(* IEC 61131-3 sources: xpxp/llama3-8b, 17 files *)

(* ---- 15.st ---- *)
FUNCTION FC1002 :BOOL
VAR_INPUT
	E_A, SENSOR: BOOL;
	ZEITW: TIME;
END_VAR
VAR
	zeit := 0;
END_VAR
VAR_IN_OUT
	ZEIT: TON;
	P_HU, P_AL: BOOL;
END_VAR

IF E_A THEN
	IF SENSOR THEN
		zeit := TIMET#(ZEITW);
		LOOP zeit < 3000 DO
			P_HU := TRUE;
			TIMET#(ZEIT) +:= 100; // Simulate sensor update (100ms)
		REPEAT
		ELOOP
		P_AL := FALSE;
		zeit := TIMET#(ZEITW);
	END_IF
ELSIF zeit > 0 THEN
	P_AL := TRUE;
ELSE
	P_HU := FALSE;
	P_AL := FALSE;
ENDIF

(* ---- 18.st ---- *)
FUNCTION FC1003 : VOID
VAR_INPUT
    IN_R:REAL;
    IN_MAX, IN_MIN:REAL;
    OUT_MAX, OUT_MIN:REAL;
END_VAR
VAR_OUTPUT
    OUT_R:REAL;
    FEH:BOOL;
END_VAR
VAR_TEMP
    DIFF1, DIFF2:REAL;
END_VAR

OUT_R := (IN_R - IN_MIN) / (IN_MAX - IN_MIN) * (OUT_MAX - OUT_MIN) + OUT_MIN;

IF OUT_R < OUT_MIN THEN
    OUT_R := OUT_MIN;
ELSIF OUT_R > OUT_MAX THEN
    OUT_R := OUT_MAX;
END_IF;

FEH := TRUE;
END_FUNCTION;

(* ---- 19.st ---- *)
FUNCTION_BLOCK FB1005

VAR_INPUT
    START: BOOL;
    DICKE: REAL;
    V_MAX: REAL;
    V_MIN: REAL;
END_VAR

VAR_OUTPUT
    D_MAX: REAL;
    D_MIN: REAL;
    P1: BOOL;
END_VAR

VAR
    FO: BOOL;
    M_MAX: REAL;
    M_MIN: REAL;
    THICKNESS: REAL;
END_VAR

PROGRAM
    IF START THEN
        M_MAX := 0.0;
        M_MIN := 0.0;
    END_IF;

    IF DICKE > 0.0 THEN
        THICKNESS := ABS(DICKE - (V_MAX + V_MIN) / 2.0);
        IF THICKNESS > M_MAX THEN
            M_MAX := THICKNESS;
        END_IF;
        IF THICKNESS < M_MIN THEN
            M_MIN := THICKNESS;
        END_IF;
    END_IF;

    D_MAX := M_MAX;
    D_MIN := M_MIN;

    IF (M_MAX > V_MAX OR M_MIN < V_MIN) THEN
        P1 := TRUE;
    ELSE
        P1 := FALSE;
    END_IF;
END_PROGRAM.

(* ---- 20.st ---- *)
FUNCTION_BLOCK INTERLOCK
VAR_INPUT
    I1 : BOOL;
    I2 : BOOL;
    TL : TIME;
END_VAR
VAR_OUTPUT
    Q1 : BOOL;
    Q2 : BOOL;
END_VAR
VAR
    T1 : TOF;
    T2 : TOF;
    t_start : TOF;
    time_count : INT := 0;
END_VAR

DO
    IF NOT I1 AND NOT T1 THEN
        T1 := #t;
    END_IF;

    IF NOT I2 AND NOT T2 THEN
        T2 := #t;
    END_IF;

    IF I1 AND NOT T1 THEN
        t_start := #t;
        time_count := 0;
    END_IF;

    IF I2 AND NOT T2 THEN
        t_start := #t;
        time_count := 0;
    END_IF;

    IF I1 AND (T1 - t_start >= TL) AND NOT Q2 THEN
        Q1 := TRUE;
        T1 := #t;
        time_count := 0;
    END_IF;

    IF I2 AND (T2 - t_start >= TL) AND NOT Q1 THEN
        Q2 := TRUE;
        T2 := #t;
        time_count := 0;
    END_IF;

    IF NOT I1 AND Q1 THEN
        T1 := #t;
    END_IF;

    IF NOT I2 AND Q2 THEN
        T2 := #t;
    END_IF;

    IF (I1 OR I2) AND (time_count > 0) THEN
        time_count := time_count - 1;
    END_IF;

END_DO;

(* ---- 21.st ---- *)
FUNCTION_BLOCK BURNER
VAR_INPUT
    IN : BOOL;
    STAGE2 : BOOL;
    OVER_TEMP : BOOL;
    OIL_TEMP : BOOL := TRUE;
    FLAME : BOOL;
    RST : BOOL;
    RST_TIMER : BOOL;
    PRE_HEAT_TIME : TIME := t#5s;
    PRE_VENT_TIME : TIME := t#15s;
    PRE_IGNITE_TIME : TIME := t#15s;
    POST_IGNITE_TIME : TIME := t#25s;
    STAGE2_DELAY : TIME := t#10s;
    SAFETY_TIME : TIME := t#5s;
    LOCKOUT_TIME : TIME := t#10s;
    MULTIPLE_IGNITION : BOOL := TRUE;
    KW1 : REAL;
    KW2 : REAL;
END_VAR
VAR_OUTPUT
    MOTOR : BOOL;
    COIL1 : BOOL;
    COIL2 : BOOL;
    PRE_HEAT : BOOL;
    IGNITE : BOOL;
    FAIL : BOOL;
    KWH : REAL;
    STATUS : BYTE;
END_VAR
VAR_IN_OUT
    RUNTIME1 : UDINT;
    RUNTIME2 : UDINT;
    CYCLES : UDINT;
END_VAR
VAR
    state : INT := 110; // standby
    last : TIME;
    tx : TIME;
    last_change : TIME;
    timer1 : TON;
    timer2 : TON;
    oil_temp_last : BOOL;
    cycles2 : UDINT;
END_VAR

PROGRAM
BEGIN
    PRE_HEAT := FALSE;
    IGNITE := FALSE;
    MOTOR := FALSE;
    COIL1 := FALSE;
    COIL2 := FALSE;
    FAIL := FALSE;
    KWH := 0;

    WHILE TRUE DO
        IF NOT OVER_TEMP AND IN THEN
            state := 111; // startup sequence
            PRE_HEAT := TRUE;
            timer1 := t#0s;
        END_IF;

        IF PRE_HEAT AND OIL_TEMP THEN
            state := 112; // burner runs on stage 1
            MOTOR := TRUE;
            timer2 := t#0s;
        END_IF;

        IF NOT FLAME AND timer2 > PRE_VENT_TIME THEN
            FAIL := TRUE;
            STATUS := 3;
        END_IF;

        IF FLAME AND timer1 > SAFETY_TIME THEN
            FAIL := TRUE;
            STATUS := 4;
        END_IF;

        IF RST THEN
            state := 110; // standby
            last_change := t#0s;
        END_IF;

        IF NOT OVER_TEMP AND RST_TIMER AND timer2 > LOCKOUT_TIME THEN
            state := 110; // standby
            last_change := t#0s;
        END_IF;

        IF MULTIPLE_IGNITION AND FLAME THEN
            IGNITE := TRUE;
            timer1 := t#0s;
        END_IF;

        IF STAGE2 AND state = 112 THEN
            state := 113; // burner runs at stage 2
            COIL2 := TRUE;
        END_IF;

        IF NOT FLAME AND timer1 > POST_IGNITE_TIME THEN
            IGNITE := FALSE;
            MOTOR := FALSE;
            COIL1 := FALSE;
            COIL2 := FALSE;
        END_IF;

    END_WHILE;

END_PROGRAM;

(* ---- 5.st ---- *)
VAR
    Start_Loop : BOOL := FALSE;
    one_hour : TIME := T#1h;
    One_Hour_Timer : TON;
    Gate_Open : BOOL := FALSE;
    Close_Gate_Inst : BOOL := FALSE;
    Sensed_Car : BOOL := FALSE;
    Sensed_Car_Inst : BOOL := FALSE;
    Sensed_App : BOOL := FALSE;
    Mobile_Inst : BOOL := FALSE;
    Auth : STRING;
    my_defined_str : STRING := 'abcd';
END_VAR

FUNCTION_BLOCK Gate_Controller

VAR_INPUT
    Start_Loop_IN : BOOL;
    Sensed_Car_IN : BOOL;
    Sensed_App_IN : BOOL;
    Mobile_IN : BOOL;
    Auth_IN : STRING;
END_VAR

VAR_OUTPUT
    Gate_Open_OUT : BOOL;
END_VAR

PROGRAM
BEGIN
    IF NOT Start_Loop THEN
        One_Hour_Timer := TON(one_hour);
    END_IF;

    IF One_Hour_Timer then
        Close_Gate_Inst := TRUE;
    END_IF;

    IF Gate_Open AND (Sensed_Car OR Sensed_App) THEN
        Auth := Auth_IN;
    END_IF;

    IF Gate_Open AND (Auth = my_defined_str) THEN
        Gate_Open_OUT := TRUE;
    ELSIF Close_Gate_Inst THEN
        Gate_Open_OUT := FALSE;
    ELSE
        Gate_Open_OUT := Gate_Open;
    END_IF;

END_PROGRAM

(* ---- 1.st ---- *)
VAR
	xAllOn : BOOL;
	xAllOff : BOOL;
	xAlarm1 : BOOL;
	xAlarm2 : BOOL;
END_VAR

PROGRAM
	IF (xAllOn) THEN
		xAlarm1 := TRUE;
		xAlarm2 := TRUE;
	END_IF;

	IF (xAllOff) THEN
		xAlarm1 := FALSE;
		xAlarm2 := FALSE;
	END_IF;
END_PROGRAM;

(* ---- 10.st ---- *)
PROGRAM SigmoidFB;

VAR
  x : REAL;
  y : REAL;
  e : REAL;
  p : REAL;

VAR_INPUT
  X : REAL;
END_VAR;

BEGIN
  e := exp(-X);
  p := 1 / (1 + e);
  y := 4.9 * p - 2.5;
END_PROGRAM;

(* ---- 11.st ---- *)
PROGRAM SignFunc;

VAR
    x : REAL;
    sign_x : REAL;
BEGIN
    IF x > 0 THEN
        sign_x := x
    ELSE
        IF x < 0 THEN
            sign_x := -x
        ELSE
            sign_x := 0;
    END_IF;
END_PROGRAM;

(* ---- 12.st ---- *)
VAR
    X : REAL;
END_VAR

VAR_OUTPUT
    Y : REAL;
END_VAR

VAR
    half_pi : REAL := 1.5707963267948966; // approximation of pi/2
    factor : REAL;
END_VAR

PROGRAM HyperbolicSine
BEGIN
    IF X < -100 OR X > 100 THEN
        Y := 0; // output is undefined for extreme values
    ELSE
        factor := exp(2 * half_pi * X);
        Y := (exp(X) - factor) / (exp(X) + factor);
    END_IF;
END_PROGRAM

(* ---- 13.st ---- *)
VAR
    nCnt : INT;
    nMaxNumber : UINT := 99;
    nSelectedNumber : INT;
    bFound : BOOL;
END_VAR

VAR_INPUT
    aNumbers : ARRAY[0..nMaxNumber] OF INT;
END_VAR

VAR_OUTPUT
    nSelectedNumber : INT;
    bFound : BOOL;
END_VAR

DO
    nCnt := 0;
    bFound := FALSE;

    REPEAT
        IF NOT bFound THEN
            nCnt := nCnt + 1;
            IF aNumbers[nCnt] = 10 THEN
                bFound := TRUE;
                EXIT;
            END_IF;
        END_IF;

        UNTIL nCnt > nMaxNumber OR bFound;

    IF bFound THEN
        nSelectedNumber := 10;
    ELSE
        nSelectedNumber := -1; // or any other value indicating "not found"
    END_IF;
END_DO

(* ---- 14.st ---- *)
PROGRAM FC1001
VAR_INPUT
    MEW: REAL;
    SP: REAL;
    HYS: REAL;
END_VAR

VAR_IN_OUT
    OUT: BOOL;
END_VAR

VAR
    P_HYS: REAL;
END_VAR

OUT := (MEW > SP + HYS/100*SP) OR (MEW < SP - HYS/100*SP);

(* ---- 16.st ---- *)
PROGRAM Traffic_Light;

VAR
    North_green         : BOOL;
    North_yellow       : BOOL;
    North_red           : BOOL;
    East_green          : BOOL;
    East_yellow         : BOOL;
    East_red             : BOOL;
    T1                   : TON;
END_VAR

PROGRAM
BEGIN
    // Initialize all lights off
    North_green := FALSE;
    North_yellow := FALSE;
    North_red     := FALSE;
    East_green    := FALSE;
    East_yellow   := FALSE;
    East_red       := FALSE;

    T1.Preset(0);
    T1.RisingEdgeTime := 10000;

    WHILE T1.Q :=# TRUE DO
        CASE T1.T
            OF 0 TO 5000 :
                North_green := TRUE;
                North_yellow := FALSE;
                North_red     := FALSE;
                East_green    := FALSE;
                East_yellow   := FALSE;
                East_red       := TRUE;
            OF 5000 TO 5500 :
                North_green := TRUE;
                North_yellow := TRUE;
                North_red     := FALSE;
                East_green    := FALSE;
                East_yellow   := FALSE;
                East_red       := TRUE;
            OF 5500 TO 9500 :
                North_green := FALSE;
                North_yellow := FALSE;
                North_red     := TRUE;
                East_green    := TRUE;
                East_yellow   := FALSE;
                East_red       := FALSE;
            OF 9500 TO 10000 :
                North_green := FALSE;
                North_yellow := FALSE;
                North_red     := TRUE;
                East_green    := FALSE;
                East_yellow   := TRUE;
                East_red       := FALSE
        END_CASE
    END_WHILE
END_PROGRAM

(* ---- 17.st ---- *)
VAR
  aiOutside : INT;
  aiHumidity: INT;
  sShowText : STRING[80];
END_VAR

PROGRAM
  IF aiOutside < 18 THEN
    sShowText := "Cold"
  ELSIF (aiOutside >= 18) AND (aiOutside <= 25) THEN
    IF (aiHumidity >= 40) AND (aiHumidity <= 75) THEN
      sShowText := "Opt"
    ELSE
      sShowText := "Temp. OK"
    END_IF
  ELSE
    sShowText := "Hot"
  END_IF

END_PROGRAM

(* ---- 2.st ---- *)
PROGRAM BinomialCoefficient;

VAR
    n : INT;
    k : INT;
    i : INT;
    result : INT;
    binomCoeff : INT;

VAR_OUTPUT
    output : INT;

BEGIN
    IF (n < 0) OR (k < 0) THEN
        output := -1; // invalid input
    ELSIF (k > n) THEN
        output := 0; // k is greater than n, coefficient is 0
    ELSE
        binomCoeff := 1;
        FOR i FROM 0 TO k DO
            IF (k - i) < (n - i) THEN
                binomCoeff := binomCoeff * (n - i);
            ELSE
                binomCoeff := binomCoeff * ((n - i) / (i + 1));
            END_IF;
        output := binomCoeff;
    END_IF;

END_PROGRAM;

(* ---- 3.st ---- *)
PROGRAM CalculateFibonacci;

VAR_INPUT
    X : INT;
END_VAR

VAR
    t1 : DINT := 0;
    t2 : DINT := 1;
    x_tmp : INT;
END_VAR

FUNCTIOIN fib : INT
    VAR
        i : INT;
    END_VAR
    i := 0;
    WHILE i < X DO
        fib := t1 + t2;
        t1 := t2;
        t2 := fib;
        i := i + 1;
    END_WHILE
END_FUNCTION

VAR_OUTPUT
    Result : INT;
END_VAR

PROGRAM
BEGIN
    IF X > 1 THEN
        Result := fib;
    ELSEIF X = 0 OR X = 1 THEN
        Result := X;
    ELSE
        Result := -1; // invalid input
    END_IF;
END_PROGRAM;

(* ---- 4.st ---- *)
VAR
    aiLevel : INT;
    PercentLevel : UINT;
    doLow : BOOL;
    doOk : BOOL;
    doHigh : BOOL;
    doAlarm : BOOL;
END_VAR

PROGRAM FillLevelCheck
    VAR_INPUT
        level : INT
    END_VAR

    CASE
        WHEN level < 327 && level > 0 THEN
            PercentLevel := (level * 100) / 32767
        ELSE
            PercentLevel := 0
    END_CASE

    CASE
        WHEN PercentLevel <= 1 THEN
            doAlarm := TRUE
            doLow := FALSE
            doOk := FALSE
            doHigh := FALSE
        WHEN PercentLevel > 1 && PercentLevel <= 66.67 THEN
            doOk := TRUE
            doLow := FALSE
            doAlarm := FALSE
            doHigh := FALSE
        WHEN PercentLevel > 66.67 THEN
            doHigh := TRUE
            doLow := FALSE
            doOk := FALSE
            doAlarm := FALSE
    END_CASE

END_PROGRAM
